PROGRAM MAIN
VAR
END_VAR

END_PROGRAM

(* stored: Version 1.1.0.1
   POU MAIN: Id {a61f7ef3-3add-4923-bf1e-4fe77a138889} *)
